Universal Robots PolyScope program: SingularityException.urp

ProgramRoot directory=/home/ur/ursim-3.1/programs/SingularityException; kinematics=(a=[0, -0.612, -0.5723, 0, 0, 0], d=[0.1273, 0, 0, 0.16394, 0.1157, 0.0922], alpha=[1.5708, 0, 0, 1.5708, -1.5708, 0], deltaTheta=[0, 0, 0, 0, 0, 0], status=notInitialized); lastSavedInVersion=(project__name=Polyscope, major__version=3, minor__version=1, svn__revision=16916, build__date=Feb 06 2015, 15:15:00); name=SingularityException; programVersion=(project__name=PolyScope, major__version=1, minor__version=8, svn__revision=11281, build__date=Aug 07 2013, 11:50:39); robotEnvironmentFileName=default; serialNumberRobot=2014350001
  MainProgram cartesianAcceleration=1.2; cartesianSpeed=0.25; jointAcceleration=1.3962634015954636; jointSpeed=1.0471975511965976; sharedProcessMoveBlendRadius=0.025; motionType=JOINT_SPACE
    Comment commentString=the following code will be ok
    Move cartesianAcceleration=1.2; cartesianSpeed=0.25; jointAcceleration=1.3962634015954636; jointSpeed=1.0471975511965976; sharedProcessMoveBlendRadius=0.025; motionType=JOINT_SPACE
      Waypoint blendRadius=0.05; cartesianAcceleration=1.2; cartesianSpeed=0.25; jointAcceleration=1.3962634015954636; jointSpeed=1.0471975511965976; nextMotionTime=2.0; stoppoint=true; useSharedBlendParameter=true; useSharedParameters=true; outputFlangePose=(pos=(x=-0.12011308439828228, y=-0.4317631339787449, z=0.14607256151643144), rot=(x=-0.0012213596815916056, y=3.116276528481971, z=0.038891915636887354)); position=TCP in base x=-179.926 y=-606.87 z=230.789 mm, rx=-0.0012 ry=3.1163 rz=0.0389 rad; joints [-91.713, -98.956, -126.223, -46.295, 91.392, -1.776] deg; positionType=FIXED_POSITION; waypointPoseInFeatureCoordinates=(pos=(x=-0.17992579232081585, y=-0.6068697097768623, z=0.2307891580793359), rot=(x=-0.001221359681589673, y=3.1162765284819924, z=0.03889191563688722)); name=Low
      Assignment expr=get_target_tcp_pose(); operatorValueType=INTEGER; valueSource=EXPRESSION
      Assignment expr=pose_add(A,p[0,0,0.5,0,0,0]); operatorValueType=INTEGER; valueSource=EXPRESSION
      Waypoint blendRadius=0.05; cartesianAcceleration=1.2; cartesianSpeed=0.25; jointAcceleration=1.3962634015954636; jointSpeed=1.0471975511965976; nextMotionTime=2.0; stoppoint=true; useSharedBlendParameter=true; useSharedParameters=true; positionType=VARIABLE_POSITION; waypointPoseInFeatureCoordinates=(pos=(x=0.0, y=0.0, z=0.0), rot=(x=0.0, y=0.0, z=0.0)); name=B_1
    Comment commentString=the following code will raise an error
    Suppressed suppressedNode=get_target_tcp_pose()
